FUNCTION_BLOCK "Delta_CFP2000"
{ S7_Optimized_Access := 'TRUE' }
VERSION : 0.1
   VAR_INPUT
      mb_addr : USInt;
      ref : Real;   // (minus rev.)
   END_VAR

   VAR_OUTPUT
      stat : Struct
         drive_stops : Bool;
         drive_decelerating : Bool;
         drive_standby : Bool;
         drive_operating : Bool;
      END_STRUCT;
      current : Real;
   END_VAR

   VAR_IN_OUT
      mb_query : "mb_query";
   END_VAR

   VAR
      s : "mb_station_udt";
      read : Struct
         warn_code : USInt;
         error_code : USInt;
         stat { ExternalAccessible := 'False'; ExternalVisible := 'False'; ExternalWritable := 'False'} : Struct
            "b08_Master frequency controlled by communication" { ExternalAccessible := 'False'; ExternalVisible := 'False'; ExternalWritable := 'False'} : Bool;
            "b09 Master frequency controlled by analog signal" { ExternalAccessible := 'False'; ExternalVisible := 'False'; ExternalWritable := 'False'} : Bool;
            "b10 Operation command controlled by communication interface" { ExternalAccessible := 'False'; ExternalVisible := 'False'; ExternalWritable := 'False'} : Bool;
            "b11 Parameter locked" { ExternalAccessible := 'False'; ExternalVisible := 'False'; ExternalWritable := 'False'} : Bool;
            "b12 Enable to copy parameters from keypad" { ExternalAccessible := 'False'; ExternalVisible := 'False'; ExternalWritable := 'False'} : Bool;
            b13 { ExternalAccessible := 'False'; ExternalVisible := 'False'; ExternalWritable := 'False'} : Bool;
            b14 { ExternalAccessible := 'False'; ExternalVisible := 'False'; ExternalWritable := 'False'} : Bool;
            b15 { ExternalAccessible := 'False'; ExternalVisible := 'False'; ExternalWritable := 'False'} : Bool;
            b00_oper_stat { ExternalAccessible := 'False'; ExternalVisible := 'False'; ExternalWritable := 'False'} : Bool;
            b01_oper_stat { ExternalAccessible := 'False'; ExternalVisible := 'False'; ExternalWritable := 'False'} : Bool;
            b02 { ExternalAccessible := 'False'; ExternalVisible := 'False'; ExternalWritable := 'False'} : Bool;
            b03_direction { ExternalAccessible := 'False'; ExternalVisible := 'False'; ExternalWritable := 'False'} : Bool;
            b04_direction { ExternalAccessible := 'False'; ExternalVisible := 'False'; ExternalWritable := 'False'} : Bool;
            b05 { ExternalAccessible := 'False'; ExternalVisible := 'False'; ExternalWritable := 'False'} : Bool;
            b06 { ExternalAccessible := 'False'; ExternalVisible := 'False'; ExternalWritable := 'False'} : Bool;
            b07 { ExternalAccessible := 'False'; ExternalVisible := 'False'; ExternalWritable := 'False'} : Bool;
         END_STRUCT;
         frequency_cmd : Int;
         output_frequency : Int;
         output_current : UInt;
         "DC-BUS Voltage" : UInt;
         output_voltage : UInt;
         "Current step number of Multi-Step Speed Operation" : Int;
         "_" : Int;
         counter_value : Int;
         power_factor_angle : Int;
         output_torque : Int;
         actual_motor_speed : Int;
         "__" : Int;
         "___" : Int;
         power_output : Int;   // kwh
      END_STRUCT;
      write { ExternalAccessible := 'False'; ExternalVisible := 'False'; ExternalWritable := 'False'} : Struct
         cmd_word { ExternalAccessible := 'False'; ExternalVisible := 'False'; ExternalWritable := 'False'} : Struct
            b08_sel_speed { ExternalAccessible := 'False'; ExternalVisible := 'False'; ExternalWritable := 'False'} : Bool;
            b09_sel_speed { ExternalAccessible := 'False'; ExternalVisible := 'False'; ExternalWritable := 'False'} : Bool;
            b10_sel_speed { ExternalAccessible := 'False'; ExternalVisible := 'False'; ExternalWritable := 'False'} : Bool;
            b11_sel_speed { ExternalAccessible := 'False'; ExternalVisible := 'False'; ExternalWritable := 'False'} : Bool;
            b12_Enable_bit06_11_function { ExternalAccessible := 'False'; ExternalVisible := 'False'; ExternalWritable := 'False'} : Bool := true;
            b13_oper_keypad { ExternalAccessible := 'False'; ExternalVisible := 'False'; ExternalWritable := 'False'} : Bool;
            b14_oper_Pr_00_21_setting { ExternalAccessible := 'False'; ExternalVisible := 'False'; ExternalWritable := 'False'} : Bool;
            b15 { ExternalAccessible := 'False'; ExternalVisible := 'False'; ExternalWritable := 'False'} : Bool;
            b00_stop { ExternalAccessible := 'False'; ExternalVisible := 'False'; ExternalWritable := 'False'} : Bool;
            b01_run { ExternalAccessible := 'False'; ExternalVisible := 'False'; ExternalWritable := 'False'} : Bool;
            b02 { ExternalAccessible := 'False'; ExternalVisible := 'False'; ExternalWritable := 'False'} : Bool;
            b03 { ExternalAccessible := 'False'; ExternalVisible := 'False'; ExternalWritable := 'False'} : Bool;
            b04_fwd { ExternalAccessible := 'False'; ExternalVisible := 'False'; ExternalWritable := 'False'} : Bool;
            b05_rev { ExternalAccessible := 'False'; ExternalVisible := 'False'; ExternalWritable := 'False'} : Bool;
            b06_sel_accel_decel { ExternalAccessible := 'False'; ExternalVisible := 'False'; ExternalWritable := 'False'} : Bool;
            b07_sel_accel_decel { ExternalAccessible := 'False'; ExternalVisible := 'False'; ExternalWritable := 'False'} : Bool;
         END_STRUCT;
         ref_freq { ExternalAccessible := 'False'; ExternalVisible := 'False'; ExternalWritable := 'False'} : UInt;
         a { ExternalAccessible := 'False'; ExternalVisible := 'False'; ExternalWritable := 'False'} : Struct
            b08 { ExternalAccessible := 'False'; ExternalVisible := 'False'; ExternalWritable := 'False'} : Bool;
            b09 { ExternalAccessible := 'False'; ExternalVisible := 'False'; ExternalWritable := 'False'} : Bool;
            b10 { ExternalAccessible := 'False'; ExternalVisible := 'False'; ExternalWritable := 'False'} : Bool;
            b11 { ExternalAccessible := 'False'; ExternalVisible := 'False'; ExternalWritable := 'False'} : Bool;
            b12 { ExternalAccessible := 'False'; ExternalVisible := 'False'; ExternalWritable := 'False'} : Bool;
            b13 { ExternalAccessible := 'False'; ExternalVisible := 'False'; ExternalWritable := 'False'} : Bool;
            b14 { ExternalAccessible := 'False'; ExternalVisible := 'False'; ExternalWritable := 'False'} : Bool;
            b15 { ExternalAccessible := 'False'; ExternalVisible := 'False'; ExternalWritable := 'False'} : Bool;
            b00_external_fault { ExternalAccessible := 'False'; ExternalVisible := 'False'; ExternalWritable := 'False'} : Bool;
            b01_reset { ExternalAccessible := 'False'; ExternalVisible := 'False'; ExternalWritable := 'False'} : Bool;
            b02_B_B_ON { ExternalAccessible := 'False'; ExternalVisible := 'False'; ExternalWritable := 'False'} : Bool;
            b03 { ExternalAccessible := 'False'; ExternalVisible := 'False'; ExternalWritable := 'False'} : Bool;
            b04 { ExternalAccessible := 'False'; ExternalVisible := 'False'; ExternalWritable := 'False'} : Bool;
            b05 { ExternalAccessible := 'False'; ExternalVisible := 'False'; ExternalWritable := 'False'} : Bool;
            b06 { ExternalAccessible := 'False'; ExternalVisible := 'False'; ExternalWritable := 'False'} : Bool;
            b07 { ExternalAccessible := 'False'; ExternalVisible := 'False'; ExternalWritable := 'False'} : Bool;
         END_STRUCT;
      END_STRUCT;
   END_VAR

   VAR_TEMP
      a : Struct
         b08 : Bool;
         b09 : Bool;
         b10 : Bool;
         b11 : Bool;
         b12 : Bool;
         b13 : Bool;
         b14 : Bool;
         b15 : Bool;
         b0 : Bool;
         b01 : Bool;
         b02 : Bool;
         b03 : Bool;
         b04 : Bool;
         b05 : Bool;
         b06 : Bool;
         b07 : Bool;
      END_STRUCT;
   END_VAR


BEGIN
	// Delta - CFP2000 - Variable frequency drive
	//
	// http://www.softstartuk.com/wp-content/uploads/2017/07/VFD-CFP2000_UM_EN_20170303.pdf

	"mb_station_header"(station := #s, mb_query := #mb_query);
	#mb_query.mb_addr := #mb_addr;

	// Read
	#mb_query.mode := #mb_query.c.read.holding_reg;

	#mb_query(data_addr := 16#2100, data_ptr := #read);
	#stat.drive_stops := NOT #read.stat.b00_oper_stat AND NOT #read.stat.b01_oper_stat;
	#stat.drive_decelerating := #read.stat.b00_oper_stat AND NOT #read.stat.b01_oper_stat;
	#stat.drive_standby := NOT #read.stat.b00_oper_stat AND #read.stat.b01_oper_stat;
	#stat.drive_operating := #read.stat.b00_oper_stat AND #read.stat.b01_oper_stat;
	#current := UINT_TO_REAL(#read.output_current) * 100;
	// Output current (XX.XX A). When current is higher than
	// 655.35, it will shift decimal as (XXX.XA). The decimal
	// can refer to High byte of 211F.

	// Write
	#mb_query.mode := #mb_query.c.write.holding_reg;

	#write.ref_freq := REAL_TO_UINT(#ref * 100);
	#write.cmd_word.b00_stop := #ref = 0;
	#write.cmd_word.b01_run := NOT #write.cmd_word.b00_stop;
	#write.cmd_word.b05_rev := #ref < 0;
	#write.cmd_word.b04_fwd := NOT #write.cmd_word.b05_rev;
	#mb_query(data_addr := 16#2000, data_ptr := #write);

	"mb_station_footer"(station := #s, mb_query := #mb_query);

END_FUNCTION_BLOCK
